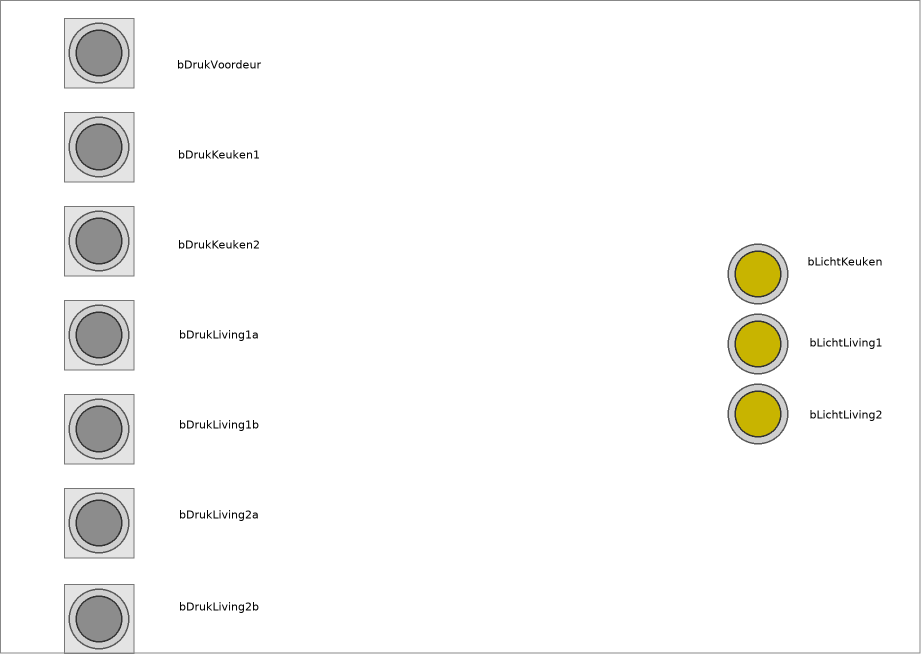
VISUALIZATION Visu  // 921x654
    PushSwitch (64,18 70x70), variable: MAIN.bDrukVoorduer, behaviour: TAP, style: Switch-PushSwitch-Gray
    PushSwitch (64,584 70x70), variable: MAIN.bDrukLiving2b, behaviour: TAP, style: Switch-PushSwitch-Gray
    PushSwitch (64,488 70x70), variable: MAIN.bDrukLiving2a, behaviour: TAP, style: Switch-PushSwitch-Gray
    PushSwitch (64,112 70x70), variable: MAIN.bDrukKeuken1, behaviour: TAP, style: Switch-PushSwitch-Gray
    PushSwitch (64,206 70x70), variable: MAIN.bDrukKeuekn2, behaviour: TAP, style: Switch-PushSwitch-Gray
    PushSwitch (64,300 70x70), variable: MAIN.bDrukLiving1a, behaviour: TAP, style: Switch-PushSwitch-Gray
    PushSwitch (64,394 70x70), variable: MAIN.bDrukLiving1b, behaviour: TAP, style: Switch-PushSwitch-Gray
    Lamp1 (723,239 70x70), variable: MAIN.bLichtKeueken, style: Lamp-Lamp1-Yellow
    Lamp1 (723,309 70x70), variable: MAIN.bLichtLiving1, style: Lamp-Lamp1-Yellow
    Lamp1 (723,379 70x70), variable: MAIN.bLichtLiving2, style: Lamp-Lamp1-Yellow
    Label (144,320 150x30), "bDrukLiving1a"
    Label (770,247 150x30), "bLichtKeuken"
    Label (144,140 150x30), "bDrukKeuken1"
    Label (144,230 150x30), "bDrukKeuken2"
    Label (144,592 150x30), "bDrukLiving2b"
    Label (144,410 150x30), "bDrukLiving1b"
    Label (144,500 150x30), "bDrukLiving2a"
    Label (144,50 150x30), "bDrukVoordeur"
    Label (771,328 150x30), "bLichtLiving1"
    Label (771,400 150x30), "bLichtLiving2"
END_VISUALIZATION

(* stored: Version 1.1.0.1, ProductVersion 3.1.4024.12
   Visu Visu: Id {f44729ab-2f4d-42e0-b489-50455d5f5b26} *)
